{attribute 'qualified_only'}
{attribute 'strict'}
TYPE E_Z6_Step :
(
	(* special steps *)
	NoStep := -32767,		// nessuno step
	Unknown := -32000,		// step sconosciuto
	
	(* Error steps *)
	NeOrError := -990,		// non abilitata o in errore
	Recovering := -980,		// azzeramento errori
		
	(* Stop *)
	Stop := 0,				// S0, stop
	
	(* Cycle *)
	Ready := 100,			// S1, pronto a ricevere pezzo
	Loading := 120,			// S2, trasferimento pezzo verso I9
	WaitUnloading := 140,	// S3, attesa rimozione pezzo da piattaforma scarico 

	Done := 800,			// Ciclo concluso
	
	(* Stopping *)
	Stopping := 900	
);
END_TYPE
//  NoStep = '-32767'
//  Unknown = '-32000'
//  NeOrError = '-990'
//  Recovering = '-980'

(* stored: Version 1.1.0.1
   EnumerationTextList E_Z6_Step: Id {f887b320-0a75-0897-0dd5-63476c78a596} *)
